(*

.. <legal notes>

legal notes
=================
| SPDX-FileCopyrightText: © 2026 Oleksandr Tiutyk <trofimich@gmail.com>
| SPDX-License-Identifier: LGPL-3.0-only
| For details check: LGPL-3.0-only_

.. _LGPL-3.0-only: https://www.gnu.org/licenses/lgpl-3.0.en.html

.. </legal notes>

*)

FUNCTION_BLOCK ABSTRACT OutputDevice EXTENDS LeafAutomationComponent IMPLEMENTS IOutputDevice

METHOD PROTECTED ABSTRACT OnProcessOutput
END_METHOD

METHOD FINAL ProcessOutput
VAR
	exceptionCode : __SYSTEM.ExceptionCode;
	exception : TOF_Core.IException;
	exceptionReaction : TOF_Core.EXCEPTION_REACTION;
END_VAR
__TRY
	OnProcessOutput();
__CATCH(exceptionCode)		
	exception := TOF_Core.ExceptionManager.GetLastException(exceptionCode);
					
	exceptionReaction := OnHandleException(exception, 'OnProcessOutput');

	ProcessException(exception, exceptionReaction, "OnProcessOutput error");
__ENDTRY
END_METHOD

END_FUNCTION_BLOCK

(* stored: Version 1.1.0.1
   POU OutputDevice: Id {105b6dfa-d76f-4477-807a-cf1396dca32a}, SpecialFunc None
   Folder Methods to override: Id {79900fc6-701a-41aa-8938-d0017f4e6cae}
   Method OnProcessOutput: Id {041a293e-47c2-48cc-bc87-e724beae058b}
   Method ProcessOutput: Id {e860c3bd-fe5d-4af5-8b65-0b4dfced7747} *)
